// Mitsubishi GX Works2 project: Counter   PLC: Q03UDV

PROGRAM MAIN
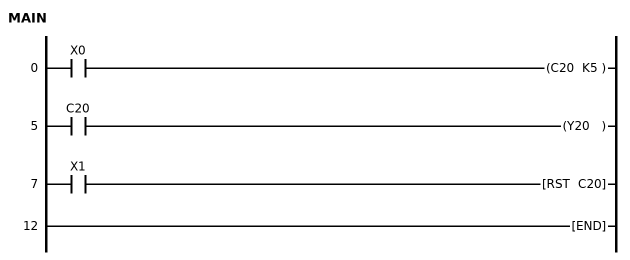
0     LD      X0
      OUT     C20 K5
5     LD      C20
      OUT     Y20
7     LD      X1
      RST     C20
12    END
END_PROGRAM
